{attribute 'pack_mode' := '1'}
TYPE ST_ChangeAxisEnable EXTENDS ST_MsgToPLC:
STRUCT
    axisIndex	: DINT;
    enabled		: BOOL;
END_STRUCT
END_TYPE

(* stored: Version 1.1.0.1, ProductVersion 3.1.4024.3
   DUT ST_ChangeAxisEnable: Id {429990be-8b42-404b-9853-8c5cb80d2e57} *)
